FUNCTION_BLOCK ObstacleChecking (* Tamplate for a simple Basic Function Block Type *)
  (* Standard: 61499-2 *)
  (* Version 0.0, 2018-10-10, 4DIAC-IDE, 4DIAC-Consortium *)
  (* Version 1.0, 2016-05-26, AZ, fortiss GmbH *)
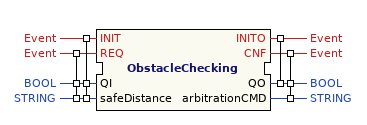
  EVENT_INPUT
    INIT WITH QI, safeDistance; (* Initialization Request *)
    REQ WITH QI, safeDistance; (* Normal Execution Request *)
  END_EVENT
  EVENT_OUTPUT
    INITO WITH QO; (* Initialization Confirm *)
    CNF WITH QO, arbitrationCMD; (* Execution Confirmation *)
  END_EVENT
  VAR_INPUT
    QI : BOOL; (* Input event qualifier *)
    safeDistance : STRING;
  END_VAR
  VAR_OUTPUT
    QO : BOOL; (* Output event qualifier *)
    arbitrationCMD : STRING;
  END_VAR
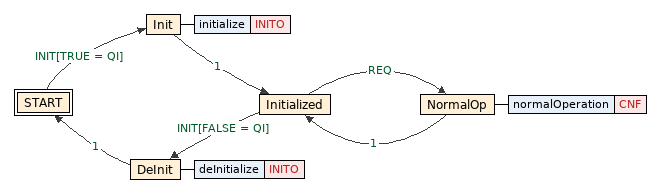
  EC_STATES
    START; (* Initial State *)
    Init : initialize -> INITO; (* Initialization *)
    NormalOp : normalOperation -> CNF; (* Normal execution *)
    Initialized;
    DeInit : deInitialize -> INITO;
  END_STATES
  EC_TRANSITIONS
    START TO Init := INIT[TRUE = QI];
    Init TO Initialized := 1;
    Initialized TO NormalOp := REQ;
    NormalOp TO Initialized := 1;
    DeInit TO START := 1;
    Initialized TO DeInit := INIT[FALSE = QI];
  END_TRANSITIONS
  ALGORITHM initialize IN ST: (* Initialization algorithm *)
QO := QI;
  END_ALGORITHM
  ALGORITHM deInitialize IN ST: (* Normally executed algorithm *)
QO := FALSE;
  END_ALGORITHM
  ALGORITHM normalOperation IN ST: (* new algorithm *)
QO := QI;

IF TRUE  = QI THEN
  (*  only perform normal operation of QI is true*)

END_IF;
  END_ALGORITHM
END_FUNCTION_BLOCK
